INTERFACE I_Datatype extends I_Serializable, I_Deserializable, I_Disposable

METHOD PUBLIC Accept
VAR_INPUT
	Visitor : I_DatatypeVisitor;
END_VAR
END_METHOD

PROPERTY PUBLIC Address : PVOID
GET
END_GET
END_PROPERTY

METHOD PUBLIC ClearReference
VAR_INPUT
END_VAR
END_METHOD

METHOD Clone : I_Datatype
END_METHOD

METHOD PUBLIC IsEquivalentTo : BOOL
VAR_INPUT
	Datatype : I_Datatype;
END_VAR
END_METHOD

PROPERTY PUBLIC IsNull : BOOL
GET
END_GET
END_PROPERTY

PROPERTY PUBLIC IsUserDefined : BOOL
GET
END_GET
END_PROPERTY

PROPERTY PUBLIC Root : I_Datatype
GET
END_GET
END_PROPERTY

METHOD PUBLIC SerializeTypeWith
VAR_INPUT
	Serializer : I_Serializer;
END_VAR
END_METHOD

PROPERTY PUBLIC Size : UDINT
GET
END_GET
END_PROPERTY

METHOD PUBLIC TryConvertTo : BOOL
VAR_INPUT
	Destination : ANY;
END_VAR
END_METHOD

METHOD PUBLIC TryConvertTo_ : BOOL
VAR_INPUT
	Destination : I_Datatype;
END_VAR
END_METHOD

METHOD PUBLIC TryCopyFrom : BOOL
VAR_INPUT
	Source : I_Datatype;
END_VAR
END_METHOD

METHOD PUBLIC ABSTRACT TryDeserializeFrom : BOOL
VAR_INPUT
	Deserializer : I_Deserializer;
	Feedback : I_DeserializerFeedback;
END_VAR
END_METHOD

METHOD TryMakeReferenceTo : BOOL
VAR_INPUT
	Target : I_Datatype;
END_VAR
END_METHOD

METHOD PUBLIC TryResolveAs_ANY : BOOL
VAR_INPUT
	Destination : REFERENCE TO I_ANY;
END_VAR
END_METHOD

METHOD PUBLIC TryResolveAs_BIT : BOOL
VAR_INPUT
	Destination : REFERENCE TO I_BIT;
END_VAR
END_METHOD

METHOD PUBLIC TryResolveAs_BOOL : BOOL
VAR_INPUT
	Destination : REFERENCE TO I_BOOL;
END_VAR
END_METHOD

METHOD PUBLIC TryResolveAs_BYTE : BOOL
VAR_INPUT
	Destination : REFERENCE TO I_BYTE;
END_VAR
END_METHOD

METHOD PUBLIC TryResolveAs_DINT : BOOL
VAR_INPUT
	Destination : REFERENCE TO I_DINT;
END_VAR
END_METHOD

METHOD PUBLIC TryResolveAs_DT : BOOL
VAR_INPUT
	Destination : REFERENCE TO I_DT;
END_VAR
END_METHOD

METHOD PUBLIC TryResolveAs_DWORD : BOOL
VAR_INPUT
	Destination : REFERENCE TO I_DWORD;
END_VAR
END_METHOD

METHOD PUBLIC TryResolveAs_INT : BOOL
VAR_INPUT
	Destination : REFERENCE TO I_INT;
END_VAR
END_METHOD

METHOD PUBLIC TryResolveAs_LINT : BOOL
VAR_INPUT
	Destination : REFERENCE TO I_LINT;
END_VAR
END_METHOD

METHOD PUBLIC TryResolveAs_LREAL : BOOL
VAR_INPUT
	Destination : REFERENCE TO I_LREAL;
END_VAR
END_METHOD

METHOD PUBLIC TryResolveAs_LWORD : BOOL
VAR_INPUT
	Destination : REFERENCE TO I_LWORD;
END_VAR
END_METHOD

METHOD PUBLIC TryResolveAs_PVOID : BOOL
VAR_INPUT
	Destination : REFERENCE TO I_PVOID;
END_VAR
END_METHOD

METHOD PUBLIC TryResolveAs_REAL : BOOL
VAR_INPUT
	Destination : REFERENCE TO I_REAL;
END_VAR
END_METHOD

METHOD PUBLIC TryResolveAs_SINT : BOOL
VAR_INPUT
	Destination : REFERENCE TO I_SINT;
END_VAR
END_METHOD

METHOD PUBLIC TryResolveAs_STRING : BOOL
VAR_INPUT
	Destination : REFERENCE TO I_STRING;
END_VAR
END_METHOD

METHOD PUBLIC TryResolveAs_TIME_OF_DAY : BOOL
VAR_INPUT
	Destination : REFERENCE TO I_TIME_OF_DAY;
END_VAR
END_METHOD

METHOD PUBLIC TryResolveAs_TOD : BOOL
VAR_INPUT
	Destination : REFERENCE TO I_TOD;
END_VAR
END_METHOD

METHOD PUBLIC TryResolveAs_UDINT : BOOL
VAR_INPUT
	Destination : REFERENCE TO I_UDINT;
END_VAR
END_METHOD

METHOD PUBLIC TryResolveAs_UINT : BOOL
VAR_INPUT
	Destination : REFERENCE TO I_UINT;
END_VAR
END_METHOD

METHOD PUBLIC TryResolveAs_ULINT : BOOL
VAR_INPUT
	Destination : REFERENCE TO I_ULINT;
END_VAR
END_METHOD

METHOD PUBLIC TryResolveAs_USINT : BOOL
VAR_INPUT
	Destination : REFERENCE TO I_USINT;
END_VAR
END_METHOD

METHOD PUBLIC TryResolveAs_WORD : BOOL
VAR_INPUT
	Destination : REFERENCE TO I_WORD;
END_VAR
END_METHOD

METHOD PUBLIC TryResolveAsAliasDatatype : BOOL
VAR_INPUT
	Destination : REFERENCE TO I_AliasDatatype;
END_VAR
END_METHOD

METHOD PUBLIC TryResolveAsArrayDatatype : BOOL
VAR_INPUT
	Destination : REFERENCE TO I_ArrayDatatype;
END_VAR
END_METHOD

METHOD PUBLIC TryResolveAsBitDatatype : BOOL
VAR_INPUT
	Destination : REFERENCE TO I_BIT;
END_VAR
END_METHOD

METHOD PUBLIC TryResolveAsEnumDatatype : BOOL
VAR_INPUT
	Destination : REFERENCE TO I_EnumDatatype;
END_VAR
END_METHOD

METHOD PUBLIC TryResolveAsInterfaceDatatype : BOOL
VAR_INPUT
	Destination : REFERENCE TO I_InterfaceDatatype;
END_VAR
END_METHOD

METHOD PUBLIC TryResolveAsStructuredDatatype : BOOL
VAR_INPUT
	Destination : REFERENCE TO I_StructuredDatatype;
END_VAR
END_METHOD

METHOD PUBLIC TryResolveAsUserDefinedDatatype : BOOL
VAR_INPUT
	Destination : REFERENCE TO I_UserDefinedDatatype;
END_VAR
END_METHOD

PROPERTY PUBLIC TypeName : T_MAXSTRING
GET
END_GET
END_PROPERTY

END_INTERFACE

(* stored: Version 1.1.0.1, ProductVersion 3.1.4026.18
   Itf I_Datatype: Id {51a69d2e-c0c1-0516-1d53-b6243b074c1e}
   Method Accept: Id {8aab0540-3d70-0faa-342b-c9c8c7ecf3f8}
   Property Address: Id {8809e202-d80e-0319-2e1b-d146d1dadc27}
   Get Get: Id {fc4214f6-2c1e-0dca-25a0-e0b18c91907f}
   Method ClearReference: Id {96eb5a41-0604-0b7a-2f4b-4cc353477151}
   Method Clone: Id {6325439c-b1ab-000e-3f25-4c490af1b6f0}
   Method IsEquivalentTo: Id {b8a569e7-18c7-0a4f-3615-23b842b124b7}
   Property IsNull: Id {ac00b9fa-f6ee-0597-1d4b-2c9f74b38274}
   Get Get: Id {dc88dfb7-140a-09ef-2d7f-b61fd3805dfe}
   Property IsUserDefined: Id {0446cf84-05ec-4e56-be5c-a67118db8177}
   Get Get: Id {30f423b3-7fa4-4d61-994e-65acaf766845}
   Property Root: Id {e7333a8b-5da9-02d2-1e69-bed566156365}
   Get Get: Id {a0608254-33d4-08b3-36e8-2c7208a013ac}
   Method SerializeTypeWith: Id {e1478293-3276-079d-0abb-6dbf50e15077}
   Property Size: Id {2ad172e6-46ce-0b59-298b-c75a14cb69e8}
   Get Get: Id {0e80b350-5013-0de5-3799-dc72c7b754fd}
   Method TryConvertTo: Id {c3e6b5b8-4372-099f-26af-6d1969bd33e8}
   Method TryConvertTo_: Id {0e70dee5-144f-0efc-127d-89c947c73ef5}
   Method TryCopyFrom: Id {d118b90b-402a-49d5-8138-4b2026e6a7a7}
   Method TryDeserializeFrom: Id {9f77e658-78c8-04ed-1f73-fb60fcdde097}
   Method TryMakeReferenceTo: Id {d965edc7-ad7d-0727-1a86-d224233b48fc}
   Method TryResolveAs_ANY: Id {34b1781a-94d0-064c-36ae-e657928ec5e7}
   Method TryResolveAs_BIT: Id {778d46eb-2742-0c97-2a64-efb935801aa5}
   Method TryResolveAs_BOOL: Id {90f66166-275f-0d22-2641-7f543ef8a66c}
   Method TryResolveAs_BYTE: Id {5aa8e4cd-2b05-0234-379f-ce01a7d54130}
   Method TryResolveAs_DINT: Id {9bf9bd26-c9eb-0206-16b7-52425ed6a222}
   Method TryResolveAs_DT: Id {36379955-d8ce-0347-0e27-3ce815b60173}
   Method TryResolveAs_DWORD: Id {9f8ba283-8fcc-044a-0590-517d836e151f}
   Method TryResolveAs_INT: Id {0c357b71-7caf-070e-2220-5f6066db843e}
   Method TryResolveAs_LINT: Id {c3d42200-4e9d-0067-0888-3311749a743f}
   Method TryResolveAs_LREAL: Id {c996eabb-6d82-06ec-2858-ccdbc458db32}
   Method TryResolveAs_LWORD: Id {0d8af125-b45b-0aac-251e-34cf0e640410}
   Method TryResolveAs_PVOID: Id {19e251cb-c110-0d33-1186-950c4ac21db5}
   Method TryResolveAs_REAL: Id {a32f2146-0000-0ec3-3f96-b23782fc82b5}
   Method TryResolveAs_SINT: Id {67cccaa3-70ca-0322-019c-66e7213071dc}
   Method TryResolveAs_STRING: Id {5ceebfa9-6cc4-02eb-30e5-d39669b76a4f}
   Method TryResolveAs_TIME_OF_DAY: Id {3d60915a-7613-0f9d-14bd-6724c077f18f}
   Method TryResolveAs_TOD: Id {5c3b4567-a014-01fd-0808-9bf48ba6973f}
   Method TryResolveAs_UDINT: Id {a4d2175d-9a02-097c-3c4e-64980ca5e865}
   Method TryResolveAs_UINT: Id {5759f2b8-840d-0b0f-357e-619e8b17a240}
   Method TryResolveAs_ULINT: Id {2afc8891-280a-03b6-1e72-b66b586a83b9}
   Method TryResolveAs_USINT: Id {ab5ca5b6-4a22-0381-045f-33f0386b545f}
   Method TryResolveAs_WORD: Id {8347f906-06c0-0055-23e6-8ec9a252f600}
   Method TryResolveAsAliasDatatype: Id {c185e5df-9218-03ac-0f52-284bc7b16735}
   Method TryResolveAsArrayDatatype: Id {74006f09-9d91-0e4d-1ae0-25993365fb62}
   Method TryResolveAsBitDatatype: Id {6cc61584-9673-045a-3102-053b316581ab}
   Method TryResolveAsEnumDatatype: Id {4f3a1c38-8ebe-03a9-1aab-375b2bf261f9}
   Method TryResolveAsInterfaceDatatype: Id {97ca1c82-d5b0-440f-8796-29491277fae6}
   Method TryResolveAsStructuredDatatype: Id {b7f6a976-614e-0340-2e42-2bb5bf32c4c6}
   Method TryResolveAsUserDefinedDatatype: Id {0efa9daa-b710-062c-3175-5c105a49bacd}
   Property TypeName: Id {42c9be80-d7dc-0e9a-0066-afba1b83ca24}
   Get Get: Id {25cf6114-32fc-0b25-2ff7-9e1b19211c00} *)
